# EPICS substitutions: mc04/tpmacApp/Db/autohome.substitutions
file "$(EPICS_BASE)/db/autohome.db"
{

pattern
{SYS,              DEV,                 PLC,  PORT  }
{"XF:23ID1-BI",  "{Diag:2-Ax:Y}",      8     P0    }
}
